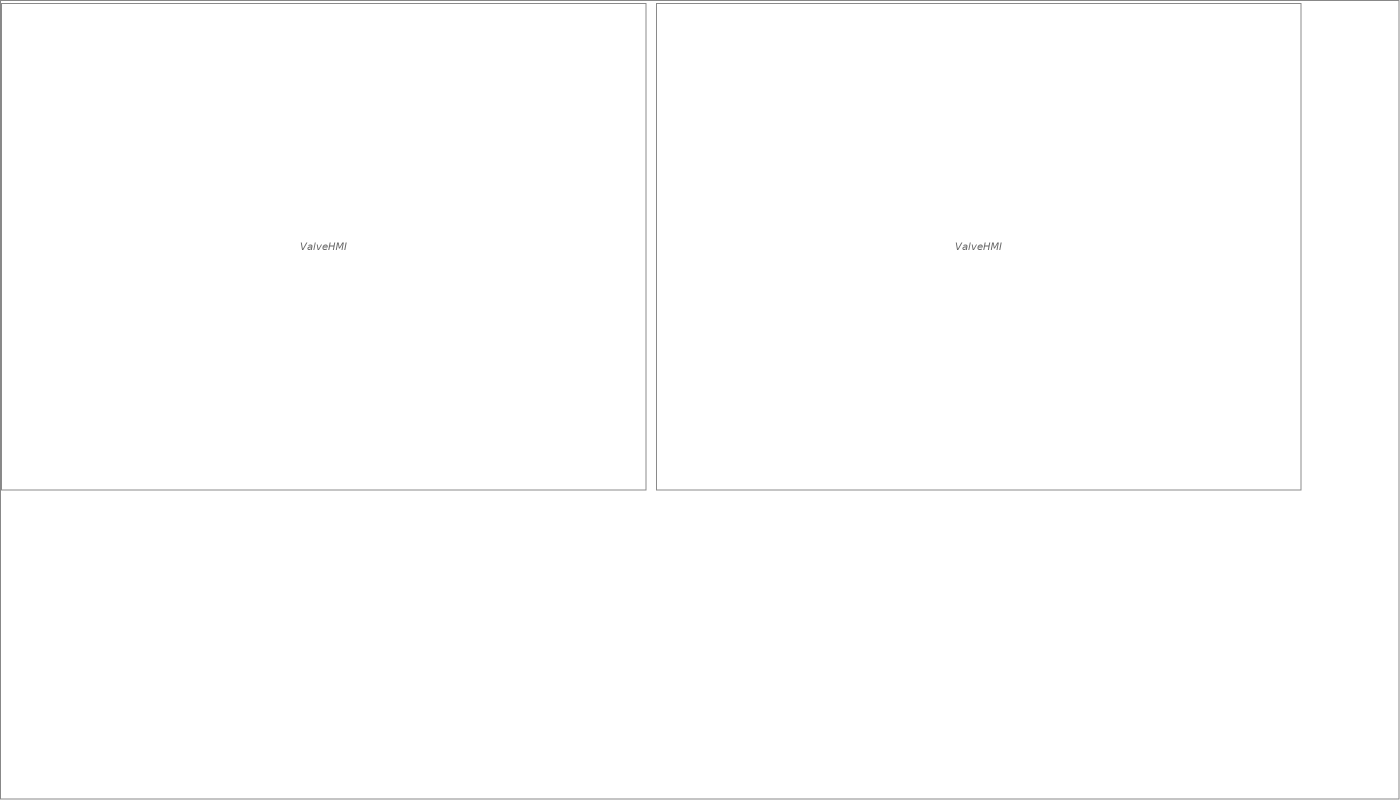
VISUALIZATION Main_Visu  // 1400x800
    Frame (1,3 645x487)
        shows ValveHMI(Valve := GVL_VCM.valve01)
    Frame (656,3 645x487)
        shows ValveHMI(Valve := GVL_VCM.valve01)
END_VISUALIZATION

(* stored: Version 1.1.0.1, ProductVersion 3.1.4024.12
   Visu Main_Visu: Id {459736cf-f2d9-4d2f-916e-a2ee046ee317} *)
